RoboDK station: RoboDK sw04a UR3e mit Robotiq First Test Hindernis Bahnplanung.rdk

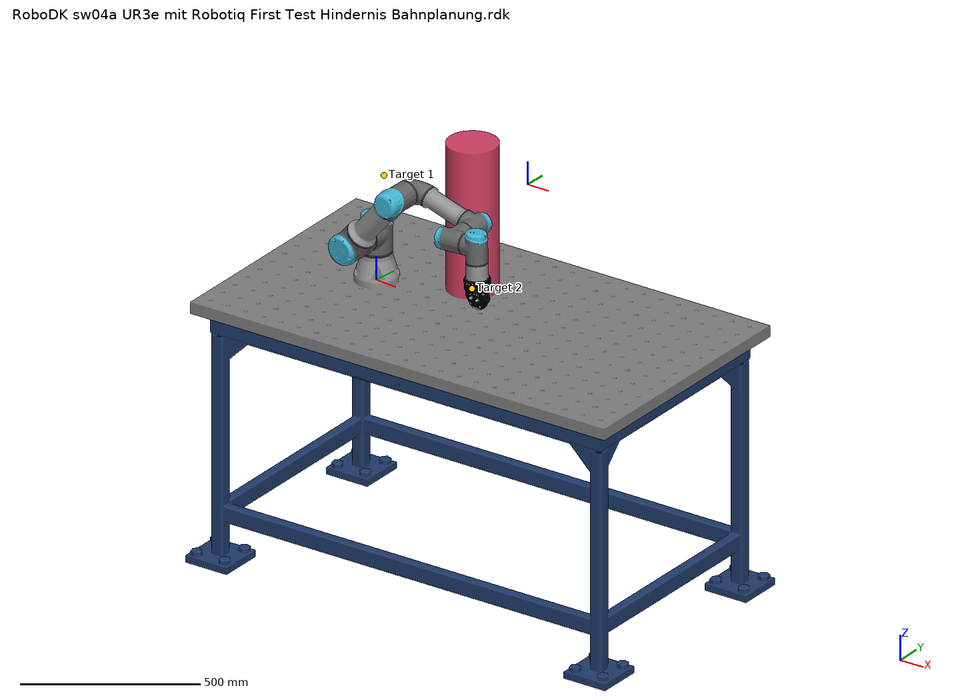
[picture v0: the station drawn from its stored meshes, robots at their saved joint values, targets as dots, program paths as lines]
Station RoboDK sw04a UR3e mit Robotiq First Test Hindernis Bahnplanung (saved by RoboDK 5.9.5). Poses are relative to the parent item; angles as X-Y-Z fixed-axis rotations.
Station parameters (name, value as stored): OPC-UA, opc.tcp://localhost:4840, CollisionFreePlanner, UR3e, CollisionFreePlanner-Rob UR3e
  - frame UR3e Base at (1.4, 12.74, 0) mm, rotated rx 0 ry 0 rz -6.26 deg
    - robot UR3e: 6 axes, payload 3 kg, reach 500 mm, repeatability 0.03 mm, weight 11 kg
        modified DH rows (alpha deg, a mm, theta deg, d mm): 0, 0, 0, 151.9; 90, 0, 180, 0; 0, 243.55, 0, 0; 0, 213.2, 0, 131.05; -90, 0, 0, 85.35; 90, 0, 180, 92.1
        joint limits [-360, -200, -360, -360, -360, -360] to [360, 27, 360, 360, 360, 360]; home [0, -90, -90, 0, 90, 0]; saved at [3.955, -130.142, -65.9, -70.622, 87.792, -80.456]
      - robot RobotiQ 2F-85 Gripper (Mechanism) (model RobotiQ 2F85): 1 axes, payload 5 kg
          joint limits [0] to [85]; home [85]; saved at [85]
        - tool Tool 1, TCP at (101.41, -36.92, 390.77) mm, rotated rx 0 ry -80.63 rz 0 deg
  - object Table 1400x800x800mm at (0, 0, 0) mm, size 1420 x 820 x 800 mm, geometry from Table-1400x800x800mm.sld
    - object Cylinder 150x450mm at (250, 120, 0) mm, size 150 x 150 x 450 mm, geometry from Cylinder-150x450mm.sld
  - frame RobotiQ 2F-85 Gripper (Mechanism) Base at (0, 742.73, 0) mm
    - target Target 1 (Cartesian target) at (-175.78, -442.67, 157.02) mm, rotated rx 177.75 ry -0.24 rz -93.37 deg; joints [150.345, -105.137, -116.115, -46.981, 91.414, 147.483] of UR3e
    - target Target 2 (Cartesian target) at (440.46, -894.89, 160.1) mm, rotated rx 179.08 ry 1.65 rz -6.26 deg; joints [2.077, -133.426, -66.92, -71.338, 89.14, -87.923] of UR3e
  - program Target1ToTarget2 (5 instructions, listed below)
  - program Target2ToTarget1 (5 instructions, listed below)
  - program MainSafe (2 instructions, listed below)
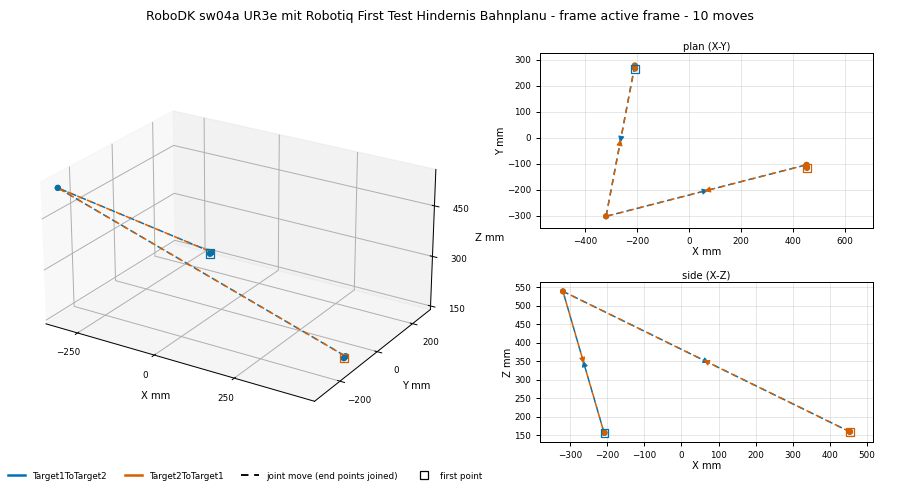
[picture p0: tool path of RoboDK sw04a UR3e mit Robotiq First Test Hindernis Bahnplanung.rdk in frame active frame, 10 of 10 moves have a stored position in this frame; points joined in program order, loops and branches not executed]

--- program Target1ToTarget2 (robot UR3e) ---
  MoveJ (Pt 1 (S18)) to (-207.45, 266.29, 157.02) mm, rotated rx 177.75 ry -0.24 rz -87.11 deg; joints [150.345, -105.137, -116.115, -46.981, 91.414, 147.483]
  MoveJ (Pt 2 (S13)) to (-208.73, 277.95, 157.02) mm, rotated rx 177.75 ry -0.24 rz -87.11 deg; joints [148.635, -107.267, -113.066, -47.944, 91.466, 145.773]
  MoveJ (Pt 3 (S74)) to (-319.51, -303.05, 538.3) mm, rotated rx 48.55 ry -5.05 rz 32.59 deg; joints [16.635, -55.232, 25.21, -72.794, 42.552, 113.879]
  MoveJ (Pt 4 (S49)) to (453.15, -104.39, 160.1) mm, rotated rx 179.08 ry 1.65 rz 0 deg; joints [3.565, -132.447, -68.704, -70.555, 89.184, -86.436]
  MoveJ (Pt 5 (S50)) to (454.43, -116.04, 160.1) mm, rotated rx 179.08 ry 1.65 rz 0 deg; joints [2.077, -133.426, -66.92, -71.338, 89.14, -87.923]

--- program Target2ToTarget1 (robot UR3e) ---
  MoveJ (Pt 1 (S50)) to (454.43, -116.04, 160.1) mm, rotated rx 179.08 ry 1.65 rz 0 deg; joints [2.077, -133.426, -66.92, -71.338, 89.14, -87.923]
  MoveJ (Pt 2 (S49)) to (453.15, -104.39, 160.1) mm, rotated rx 179.08 ry 1.65 rz 0 deg; joints [3.565, -132.447, -68.704, -70.555, 89.184, -86.436]
  MoveJ (Pt 3 (S74)) to (-319.51, -303.05, 538.3) mm, rotated rx 48.55 ry -5.05 rz 32.59 deg; joints [16.635, -55.232, 25.21, -72.794, 42.552, 113.879]
  MoveJ (Pt 4 (S13)) to (-208.73, 277.95, 157.02) mm, rotated rx 177.75 ry -0.24 rz -87.11 deg; joints [148.635, -107.267, -113.066, -47.944, 91.466, 145.773]
  MoveJ (Pt 5 (S18)) to (-207.45, 266.29, 157.02) mm, rotated rx 177.75 ry -0.24 rz -87.11 deg; joints [150.345, -105.137, -116.115, -46.981, 91.414, 147.483]

--- program MainSafe (robot UR3e) ---
  Call Target2ToTarget1
  Call Target1ToTarget2
